FUNCTION_BLOCK AR_model
  (* Version 1.0, 2005-09-21, Goran Cengic, Chalmers *)
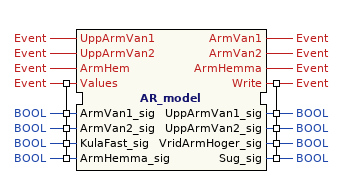
  EVENT_INPUT
    UppArmVan1;
    UppArmVan2;
    ArmHem;
    Values WITH ArmVan1_sig, ArmVan2_sig, KulaFast_sig, ArmHemma_sig;
  END_EVENT
  EVENT_OUTPUT
    ArmVan1;
    ArmVan2;
    ArmHemma;
    Write WITH UppArmVan1_sig, UppArmVan2_sig, VridArmHoger_sig, Sug_sig;
  END_EVENT
  VAR_INPUT
    ArmVan1_sig : BOOL;
    ArmVan2_sig : BOOL;
    KulaFast_sig : BOOL;
    ArmHemma_sig : BOOL;
  END_VAR
  VAR_OUTPUT
    UppArmVan1_sig : BOOL;
    UppArmVan2_sig : BOOL;
    VridArmHoger_sig : BOOL;
    Sug_sig : BOOL;
  END_VAR
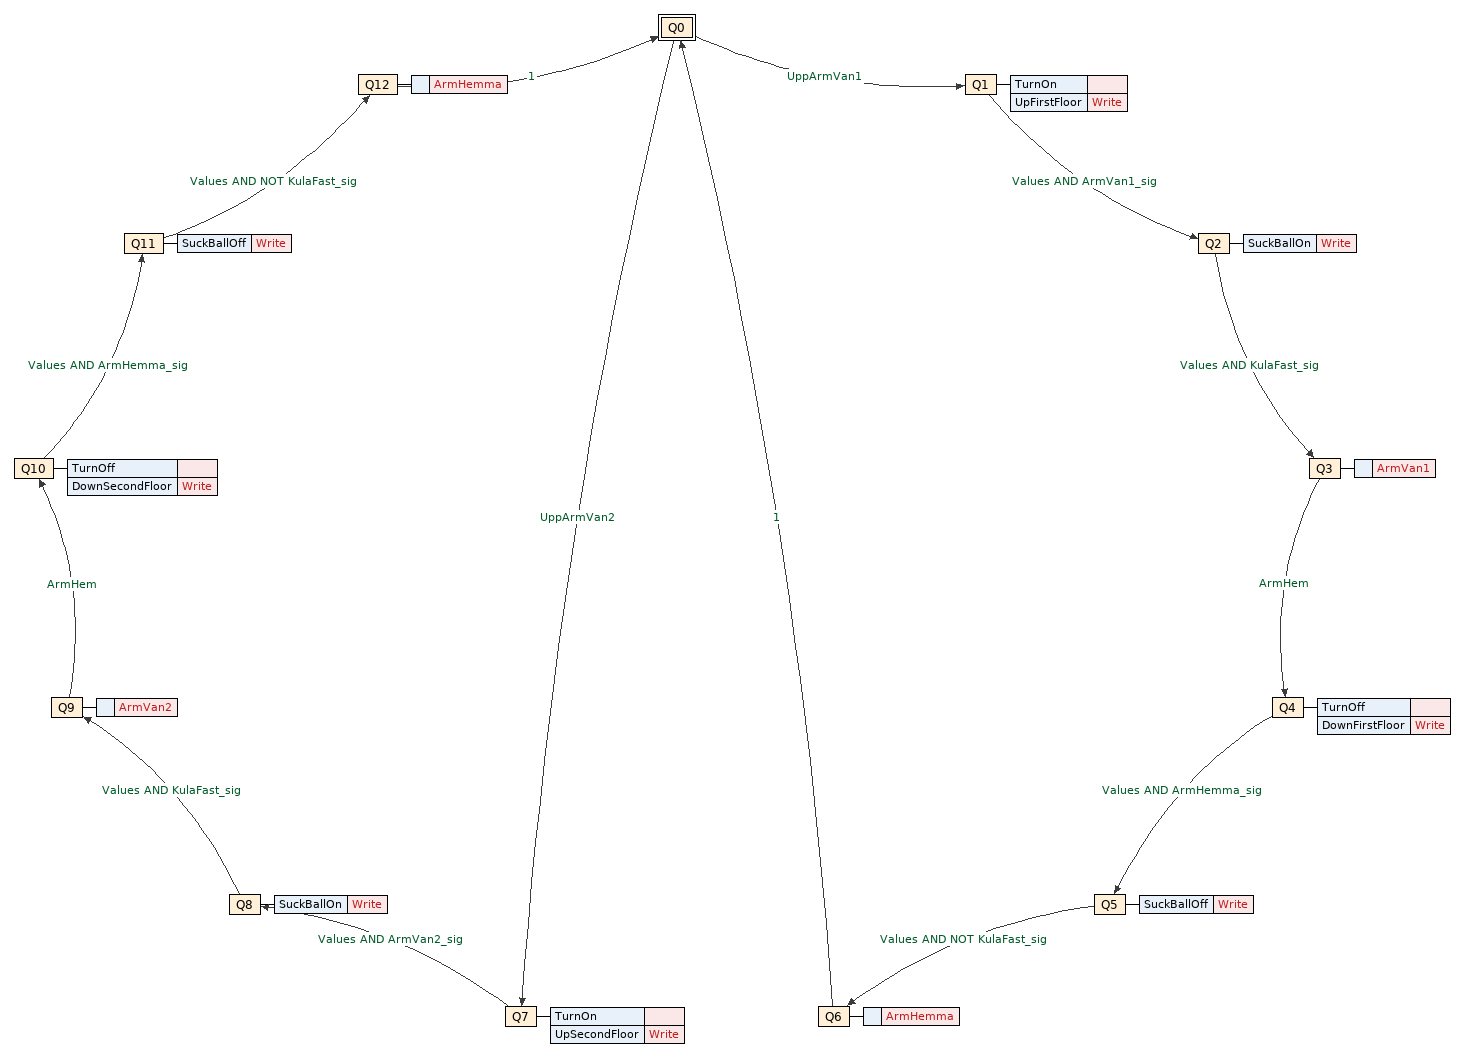
  EC_STATES
    Q0;
    Q1 : TurnOn, UpFirstFloor -> Write;
    Q2 : SuckBallOn -> Write;
    Q3 : -> ArmVan1;
    Q4 : TurnOff, DownFirstFloor -> Write;
    Q5 : SuckBallOff -> Write;
    Q6 : -> ArmHemma;
    Q7 : TurnOn, UpSecondFloor -> Write;
    Q8 : SuckBallOn -> Write;
    Q9 : -> ArmVan2;
    Q10 : TurnOff, DownSecondFloor -> Write;
    Q11 : SuckBallOff -> Write;
    Q12 : -> ArmHemma;
  END_STATES
  EC_TRANSITIONS
    Q0 TO Q1 := UppArmVan1;
    Q1 TO Q2 := Values AND ArmVan1_sig;
    Q2 TO Q3 := Values AND KulaFast_sig;
    Q3 TO Q4 := ArmHem;
    Q4 TO Q5 := Values AND ArmHemma_sig;
    Q5 TO Q6 := Values AND NOT KulaFast_sig;
    Q6 TO Q0 := 1;
    Q0 TO Q7 := UppArmVan2;
    Q7 TO Q8 := Values AND ArmVan2_sig;
    Q8 TO Q9 := Values AND KulaFast_sig;
    Q9 TO Q10 := ArmHem;
    Q10 TO Q11 := Values AND ArmHemma_sig;
    Q11 TO Q12 := Values AND NOT KulaFast_sig;
    Q12 TO Q0 := 1;
  END_TRANSITIONS
  ALGORITHM TurnOn IN Java:
		System.out.println("Arm turning right.");
		VridArmHoger_sig = true;
  END_ALGORITHM
  ALGORITHM TurnOff IN Java:
		System.out.println("Arm turning left.");
		VridArmHoger_sig = false;
  END_ALGORITHM
  ALGORITHM SuckBallOn IN Java:
		System.out.println("Arm sucking ball.");
		Sug_sig = true;
  END_ALGORITHM
  ALGORITHM SuckBallOff IN Java:
		System.out.println("Arm releasing ball.");
		Sug_sig = false;
  END_ALGORITHM
  ALGORITHM UpSecondFloor IN Java:
		System.out.println("Arm going up to second floor.");
		UppArmVan2_sig = true;
  END_ALGORITHM
  ALGORITHM DownSecondFloor IN Java:
		System.out.println("Arm going down from second floor.");
		UppArmVan2_sig = false;
  END_ALGORITHM
  ALGORITHM UpFirstFloor IN Java:
		System.out.println("Arm going up to first floor.");
		UppArmVan1_sig = true;
  END_ALGORITHM
  ALGORITHM DownFirstFloor IN Java:
		System.out.println("Arm going down from first floor.");
		UppArmVan1_sig = false;
  END_ALGORITHM
END_FUNCTION_BLOCK
